KUKA KRL program: testmain.src, testmain.dat

--- testmain.src ---
&ACCESS RVP
&REL 1
&PARAM EDITMASK = *
&PARAM TEMPLATE = C:\KRC\Roboter\Template\vorgabe
&PARAM DISKPATH = KRC:\R1\Program
DEF testmain( )
;fold FRAME
DECL FRAME READY_POS
DECL FRAME stack_POS
DECL FRAME up_pos
DECL FRAME stack_end
DECL FRAME rotation_pos
DECL INT X
;endfold
;FOLD INI;%{PE}
  ;FOLD BASISTECH INI
    GLOBAL INTERRUPT DECL 3 WHEN $STOPMESS==TRUE DO IR_STOPM ( )
    INTERRUPT ON 3
    BAS (#INITMOV,0 )
  ;ENDFOLD (BASISTECH INI)
  ;FOLD USER INI
    ;Make your modifications here

  ;ENDFOLD (USER INI)
;ENDFOLD (INI)
;FOLD PTP HOME  Vel= 100 % DEFAULT;%{PE}%MKUKATPBASIS,%CMOVE,%VPTP,%P 1:PTP, 2:HOME, 3:, 5:100, 7:DEFAULT
$BWDSTART = FALSE
PDAT_ACT=PDEFAULT
FDAT_ACT=FHOME
BAS (#PTP_PARAMS,100 )
$H_POS=XHOME
PTP  XHOME
;ENDFOLD
if false then
;FOLD PTP maduo Vel=100 % PDAT1 Tool[1] Base[1];%{PE}%R 8.3.22,%MKUKATPBASIS,%CMOVE,%VPTP,%P 1:PTP, 2:maduo, 3:, 5:100, 7:PDAT1
$BWDSTART=FALSE
PDAT_ACT=PPDAT1
FDAT_ACT=Fmaduo
BAS(#PTP_PARAMS,100)
PTP Xmaduo
;ENDFOLD
endif
loop
continue
$advance=3
;FOLD USER INI
$out[2]=FALSE
$OUT[3]=false
$OUT[4]=false
;ENDFOLD
$advance=3
;PTP Pick_Up
continue
;wait for $in[1] and $in[2] AND $aut ;wait allow Pick
;PTP Pick_pos
$ov_pro=10
$advance=3
;PTP pick_Up
;FOLD PTP pick_up CONT Vel=100 % PDAT4 Tool[1] Base[1];%{PE}%R 8.2.24,%MKUKATPBASIS,%CMOVE,%VPTP,%P 1:PTP, 2:pick_up, 3:C_DIS, 5:100, 7:PDAT4
$BWDSTART=FALSE
PDAT_ACT=PPDAT4
FDAT_ACT=Fpick_up
BAS(#PTP_PARAMS,100)
PTP Xpick_up C_DIS
;ENDFOLD
calculation()
CONTINUE
;start rotation
;START TO MADUO
;fold up_POS
up_POS=Xmaduo
up_POS.X=up_POS.X+P_POSITION[Tier,Num].X
$BASE=BASE_DATA[1]
FOR X=1 TO 6
$VEL_AXIS[X]=85
$ACC_AXIS[X]=85
ENDFOR
$APO.CPTP=5
ptp up_POS C_DIS
;endfold
;START
;fold READY_POS
READY_POS=Xmaduo
READY_POS.Z=READY_POS.Z+RH
$BASE=BASE_DATA[1]
FOR X=1 TO 6
$VEL_AXIS[X]=85
$ACC_AXIS[X]=85
ENDFOR
$APO.CPTP=5
ptp READY_POS C_DIS
;endfold
; stack start
;FOLD STACK_POS
stack_POS=Xmaduo
stack_POS.X=stack_POS.X+P_POSITION[Tier,Num].X
$BASE=BASE_DATA[1]
FOR X=1 TO 6
$VEL_AXIS[X]=85
$ACC_AXIS[X]=85
ENDFOR
$APO.CPTP=5
ptp stack_POS C_DIS
;ENDFOLD
$OUT[2]=FALSE
$OUT[4]=true
$advance=3
;STACK END
;FOLD STACK_END
stack_end=Xmaduo
stack_POS.Z=stack_POS.Z+RH
$BASE=BASE_DATA[1]
FOR X=1 TO 6
$VEL_AXIS[X]=85
$ACC_AXIS[X]=85
ENDFOR
$APO.CPTP=5
ptp stack_end C_DIS
;ENDFOLD
$out[3]=false
$out[4]=false
$ov_pro=10
;FOLD COUNT
Tier=Tier+1
if Tier==2 then
   NUM=Num+1
  tier=1
endif
if num==3 then
   num=1
goto mark
endif
;ENDFOLD
endloop
mark:
;FOLD PTP HOME  Vel= 100 % DEFAULT;%{PE}%MKUKATPBASIS,%CMOVE,%VPTP,%P 1:PTP, 2:HOME, 3:, 5:100, 7:DEFAULT
$BWDSTART = FALSE
PDAT_ACT=PDEFAULT
FDAT_ACT=FHOME
BAS (#PTP_PARAMS,100 )
$H_POS=XHOME
PTP  XHOME
;ENDFOLD
END

--- testmain.dat ---
&ACCESS RVP
&REL 1
&PARAM EDITMASK = *
&PARAM TEMPLATE = C:\KRC\Roboter\Template\vorgabe
&PARAM DISKPATH = KRC:\R1\Program
DEFDAT  testmain
;FOLD EXTERNAL DECLARATIONS;%{PE}%MKUKATPBASIS,%CEXT,%VCOMMON,%P
;FOLD BASISTECH EXT;%{PE}%MKUKATPBASIS,%CEXT,%VEXT,%P
EXT  BAS (BAS_COMMAND  :IN,REAL  :IN )
DECL INT SUCCESS
;ENDFOLD (BASISTECH EXT)
;FOLD USER EXT;%{E}%MKUKATPUSER,%CEXT,%VEXT,%P
;Make your modifications here

;ENDFOLD (USER EXT)
;ENDFOLD (EXTERNAL DECLARATIONS)
DECL BASIS_SUGG_T LAST_BASIS={POINT1[] "frist2                  ",POINT2[] "frist2                  ",CP_PARAMS[] "CPDAT0                  ",PTP_PARAMS[] "PDAT10                  ",CONT[] "                        ",CP_VEL[] "2.0                     ",PTP_VEL[] "100                     ",SYNC_PARAMS[] "SYNCDAT                 ",SPL_NAME[] "S0                      "}
DECL E6POS XMADUO={X 127.859245,Y 185.886246,Z -89.9371643,A 101.680458,B -3.80285215,C -178.452240,S 2,T 34,E1 0.0,E2 0.0,E3 0.0,E4 0.0,E5 0.0,E6 0.0}
DECL FDAT Fmaduo={TOOL_NO 1,BASE_NO 1,IPO_FRAME #BASE,POINT2[] " ",TQ_STATE FALSE}
DECL PDAT PPDAT1={VEL 100.000,ACC 100.000,APO_DIST 100.000,GEAR_JERK 50.0000}
DECL E6POS XPICK={X -102.774834,Y 251.292023,Z 361.431549,A 101.678474,B -3.80238652,C -178.452682,S 2,T 2,E1 0.0,E2 0.0,E3 0.0,E4 0.0,E5 0.0,E6 0.0}
DECL FDAT Fpick={TOOL_NO 1,BASE_NO 1,IPO_FRAME #BASE,POINT2[] " ",TQ_STATE FALSE}
DECL PDAT PPDAT2={VEL 100.000,ACC 100.000,APO_DIST 100.000,GEAR_JERK 50.0000}
DECL E6POS XPICK_UP={X -64.2057724,Y 191.421478,Z 158.514542,A 101.687286,B -3.79593801,C -178.432693,S 2,T 2,E1 0.0,E2 0.0,E3 0.0,E4 0.0,E5 0.0,E6 0.0}
DECL FDAT Fpick_up={TOOL_NO 1,BASE_NO 1,IPO_FRAME #BASE,POINT2[] " ",TQ_STATE FALSE}
DECL PDAT PPDAT3={VEL 100.000,ACC 100.000,APO_DIST 100.000,APO_MODE #CDIS,GEAR_JERK 50.0000}
DECL PDAT PPDAT4={VEL 100.000,ACC 100.000,APO_DIST 100.000,APO_MODE #CDIS,GEAR_JERK 50.0000}
DECL E6POS XFRIST={X 347.103729,Y -317.262756,Z 521.114380,A -168.321411,B -3.80309796,C -178.453552,S 2,T 2,E1 0.0,E2 0.0,E3 0.0,E4 0.0,E5 0.0,E6 0.0}
DECL FDAT Ffrist={TOOL_NO 1,BASE_NO 0,IPO_FRAME #BASE,POINT2[] " ",TQ_STATE FALSE}
DECL PDAT PPDAT5={VEL 100.000,ACC 100.000,APO_DIST 100.000,GEAR_JERK 50.0000}
DECL PDAT PPDAT6={VEL 100.000,ACC 100.000,APO_DIST 100.000,GEAR_JERK 50.0000}
DECL E6POS XFRIST1={X 4932.72314,Y 239.200607,Z 876.474487,A 120.238602,B 0.000230552105,C 180.000,S 2,T 43,E1 0.0,E2 0.0,E3 0.0,E4 0.0,E5 0.0,E6 0.0}
DECL FDAT Ffrist1={TOOL_NO 1,BASE_NO 1,IPO_FRAME #BASE,POINT2[] " ",TQ_STATE FALSE}
DECL PDAT PPDAT7={VEL 100.000,ACC 100.000,APO_DIST 100.000,GEAR_JERK 50.0000}
DECL E6POS XFRIST2={X 3538.39600,Y 2042.02905,Z 1538.35803,A -133.566101,B -0.000567811716,C -179.999802,S 2,T 11,E1 0.0,E2 0.0,E3 0.0,E4 0.0,E5 0.0,E6 0.0}
DECL FDAT Ffrist2={TOOL_NO 1,BASE_NO 1,IPO_FRAME #BASE,POINT2[] " ",TQ_STATE FALSE}
DECL PDAT PPDAT8={VEL 100.000,ACC 100.000,APO_DIST 100.000,GEAR_JERK 50.0000}
DECL E6POS Xrotation={X 3345.06812,Y 2038.01,Z 1538.40698,A -133.580795,B -0.000434641697,C -179.999603,S 2,T 11,E1 0.0,E2 0.0,E3 0.0,E4 0.0,E5 0.0,E6 0.0}
DECL FDAT Frotation={TOOL_NO 1,BASE_NO 1,IPO_FRAME #BASE,POINT2[] " ",TQ_STATE FALSE}
DECL PDAT PPDAT9={VEL 100.000,ACC 100.000,APO_DIST 100.000,GEAR_JERK 50.0000}
DECL PDAT PPDAT10={VEL 100.000,ACC 100.000,APO_DIST 100.000,GEAR_JERK 50.0000}
ENDDAT
